// TIA Portal V19 export
FUNCTION_BLOCK "A0301_Trasporto_FB"   // FB61, LAD
TITLE = == GESTIONE NASTRI TRASPORTO ==
// stored: MemoryReserve 100, SetENOAutomatically false
   VAR_INPUT
      AreaInterface : "AreaInterface";
      ZSI : "udt_ZoneSafetyInterface";
      DSI : "udt_DeviceSafetyInterface";
      Drive : "TAx_DriveInterface";
      DataIn : "SpeedMachine_DataIn";
      CIn : Struct
         Drive : "SpeedMachine_CIn";
         OP_SemiAut_PB : Bool;
      END_STRUCT;
      Config : "SpeedMachine_Config";
      HWID_Ax_TEL1 : HW_SUBMODULE;
   END_VAR
   VAR_OUTPUT
      MachineInterface { ExternalAccessible := 'False'; ExternalVisible := 'False'; ExternalWritable := 'False'} : "MachineInterface";
      COut : Struct
         Ax : "SpeedMachine_COut";
         Ax_VelOveride : Struct
            Enable : Bool;
            Value : Real;
         END_STRUCT;
      END_STRUCT;
   END_VAR
   VAR_IN_OUT
      Par : Struct
         Ax : "SpeedMachine_Par";
         Ax_Aut : "A0301_Mach_Speed_Par";
      END_STRUCT;
   END_VAR
   VAR
      Alarm : Struct
         Ax { ExternalVisible := 'False'} : "SpeedMachine_Alr";
      END_STRUCT;
      Warning : Struct
         Ax { S7_SetPoint := 'True'} : "SpeedMachine_Wng";
         OP_REST_MissingCnd : Bool;   // Mancanza comando arresto
         OP_WORK_MissingCnd : Bool;   // Mancanza consenso lavoro
      END_STRUCT;
      Ax : "SpeedMachine_FB";
      ValueVelOvr { ExternalAccessible := 'False'; ExternalVisible := 'False'; ExternalWritable := 'False'} : Array[1..10] of Real;
      Sts : Struct
         OP_CanMoveFreely : Bool;
         OP_Bwd_Cnd : Bool;
         OP_Fwd_Cnd : Bool;
      END_STRUCT;
      Ctrl : Struct
         OP_Bwd_Man : Bool;
         OP_Fwd_Man : Bool;
         OP_Bwd_Aut : Bool;
         OP_Fwd_Aut : Bool;
         OP_Bwd_Run : Bool;
         OP_Fwd_Run : Bool;
      END_STRUCT;
      AUX : Struct
         OP_Bwd_PB : Bool;
         OP_Fwd_PB : Bool;
      END_STRUCT;
      TON_OP_REST_MissingCnd { S7_SetPoint := 'True'} : TON_TIME;
      TON_OP_WORK_MissingCnd { S7_SetPoint := 'True'} : TON_TIME;
   END_VAR
   VAR_TEMP
      PE : Struct
         OP_Bwd_PB : Bool;
         OP_Fwd_PB : Bool;
      END_STRUCT;
      VelOvr_Max : Real;   // Velocità max trovata
      i : Int;
      Check : Struct
         Cndz1_StartFwd : Bool;   // Check conditions to P4
         Cndz2_StartFwd : Bool;   // Check conditions to Allineatore laterale
      END_STRUCT;
   END_VAR
   VAR_TEMP   // added for the SCL form of the ladder/FBD networks
      _w1 : Bool;
      _w2 : Bool;
      _w3 : Bool;
   END_VAR
BEGIN

REGION Network 1 (SCL): == Riferimenti [Ax] - Speed Machine ==
   // ******************************************************************************************
   REGION // TRASFERIMENTO DELLE RAMPE

       // Rampe in Manuale
       IF #AreaInterface.Man AND NOT #CIn.OP_SemiAut_PB THEN
           #Ax.CIn.Manager.Vel := #Par.Ax.Man.VelFwdHigh;
           #Ax.CIn.Manager.Acc := #Par.Ax.Man.Acc;
           #Ax.CIn.Manager.Dec := #Par.Ax.Man.Dec;
       END_IF;
   END_REGION


   // ******************************************************************************************
   REGION // CALCOLO DELLA VELOCITA' TRASFERITA DALL'IMPIANTO IN BASE ALLA LUNGHEZZA DEL PEZZO 

       // Inizializzo variabile di appoggio controllo overide massimo a un valore basso rispetto setpoint
       IF "Sys".AuxFirstPLCCycle THEN
           #VelOvr_Max := 100.0;
       END_IF;

       // Trasferisco le varibili su un array
       #ValueVelOvr[1] := "PPrf_MAIN".ON_WORK.A0301_A0302.Trasporto.VelOvr_PLen_UpTo_1000;
       #ValueVelOvr[2] := "PPrf_MAIN".ON_WORK.A0301_A0302.Trasporto.VelOvr_PLen_UpTo_1500;
       #ValueVelOvr[3] := "PPrf_MAIN".ON_WORK.A0301_A0302.Trasporto.VelOvr_PLen_UpTo_2000;
       #ValueVelOvr[4] := "PPrf_MAIN".ON_WORK.A0301_A0302.Trasporto.VelOvr_PLen_UpTo_2500;
       #ValueVelOvr[5] := "PPrf_MAIN".ON_WORK.A0301_A0302.Trasporto.VelOvr_PLen_UpTo_3000;
       #ValueVelOvr[6] := "PPrf_MAIN".ON_WORK.A0301_A0302.Trasporto.VelOvr_PLen_UpTo_3500;
       #ValueVelOvr[7] := "PPrf_MAIN".ON_WORK.A0301_A0302.Trasporto.VelOvr_PLen_UpTo_4000;
       #ValueVelOvr[8] := "PPrf_MAIN".ON_WORK.A0301_A0302.Trasporto.VelOvr_PLen_UpTo_4500;
       #ValueVelOvr[9] := "PPrf_MAIN".ON_WORK.A0301_A0302.Trasporto.VelOvr_PLen_UpTo_5000;
       #ValueVelOvr[10] := "PPrf_MAIN".ON_WORK.A0301_A0302.Trasporto.VelOvr_PLen_UpTo_5500;


       // Ciclo per verificare la variabile maggiore per prenderla in lavoro
       FOR #i := 1 TO 10 DO
           IF #ValueVelOvr[#i] >= #VelOvr_Max THEN
               #VelOvr_Max := #ValueVelOvr[#i];
           END_IF;
       END_FOR;
   END_REGION ;

   IF #VelOvr_Max = 0.0 THEN
       #VelOvr_Max := 100.0;
   END_IF;

   // ******************************************************************************************
   REGION // CALCOLO DELLA VELOCITA' E TRASFERIMENTO IN BASE ALLO STATO IMPIANTO
       #Ax.CIn.Manager := #CIn.Drive.Manager;

       IF #Ax.CIn.Manager.Control_ON THEN
           // CALCOLO VELOCITA' IN BASE ALL'OVERIDE
           IF #Ax.AreaInterface.Aut THEN
               #Ax.CIn.Manager.Vel := (#Par.Ax_Aut.Aut_Vel * #VelOvr_Max);
           END_IF;

           IF #CIn.OP_SemiAut_PB AND NOT #Ax.AreaInterface.Aut THEN
               #Ax.CIn.Manager.Vel := (#Par.Ax_Aut.SemiAut_Vel* #VelOvr_Max);
               #Ax.CIn.Manager.Acc := #Par.Ax_Aut.Aut_Acc;
               #Ax.CIn.Manager.Dec := #Par.Ax_Aut.Aut_Dec;
           END_IF;
       END_IF;
   END_REGION ;
   //


       #COut.Ax_VelOveride.Enable := TRUE;
       #COut.Ax_VelOveride.Value := #VelOvr_Max;
END_REGION

REGION Network 3: Operazione può muoversi liberamente perchè non sposta nessun BEAM
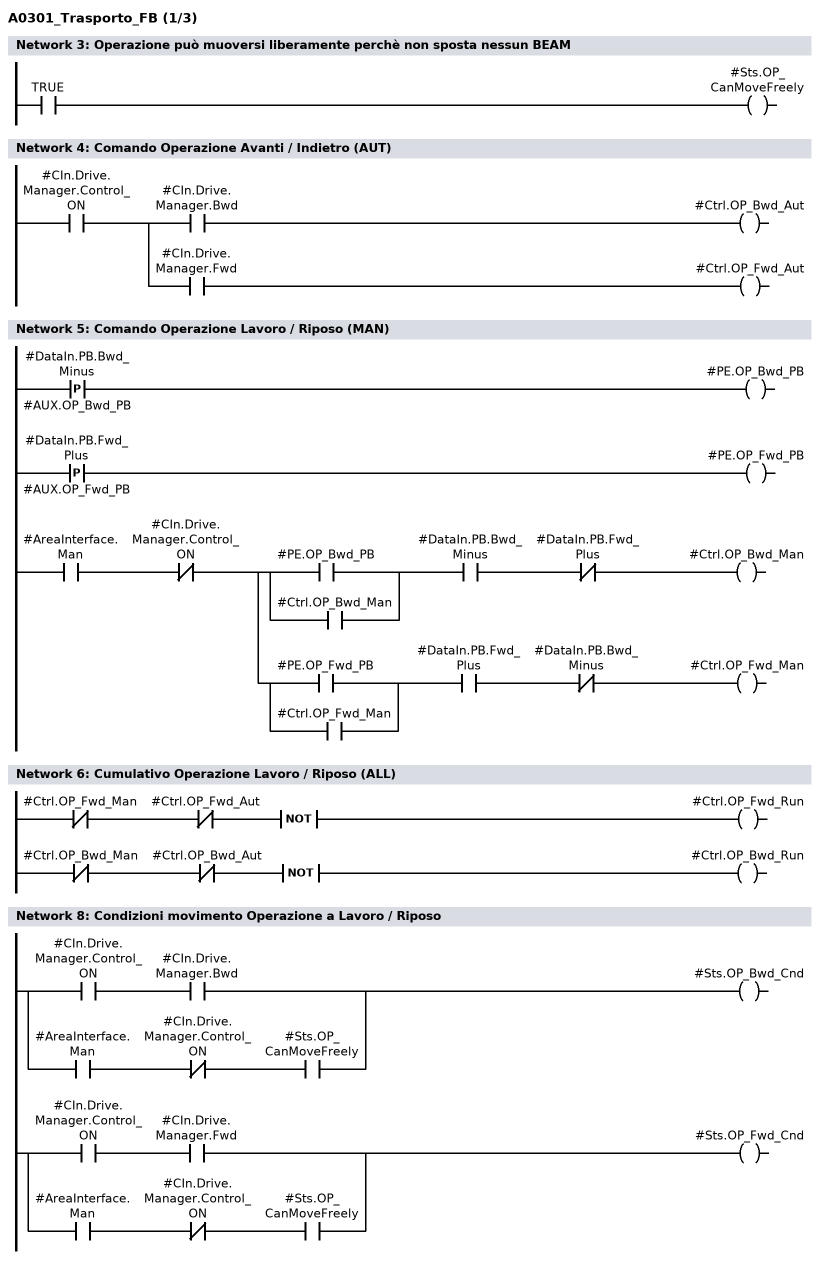
   RUNG wire#powerrail
      Contact( TRUE )
      Coil( #Sts.OP_CanMoveFreely )
   END_RUNG
   // the same network as SCL:
   #Sts.OP_CanMoveFreely := TRUE;
END_REGION

REGION Network 4: Comando Operazione Avanti / Indietro (AUT)
   RUNG wire#powerrail
      Contact( #CIn.Drive.Manager.Control_ON )
      wire#w1
      Contact( #CIn.Drive.Manager.Bwd )
      Coil( #Ctrl.OP_Bwd_Aut )
   END_RUNG
   RUNG wire#w1
      Contact( #CIn.Drive.Manager.Fwd )
      Coil( #Ctrl.OP_Fwd_Aut )
   END_RUNG
   // the same network as SCL:
   #Ctrl.OP_Bwd_Aut := #CIn.Drive.Manager.Control_ON AND #CIn.Drive.Manager.Bwd;
   #Ctrl.OP_Fwd_Aut := #CIn.Drive.Manager.Control_ON AND #CIn.Drive.Manager.Fwd;
END_REGION

REGION Network 5: Comando Operazione Lavoro / Riposo (MAN)
   RUNG wire#powerrail
      P_Contact(operand := #DataIn.PB.Bwd_Minus, bit := #AUX.OP_Bwd_PB)
      Coil( #PE.OP_Bwd_PB )
   END_RUNG
   RUNG wire#powerrail
      P_Contact(operand := #DataIn.PB.Fwd_Plus, bit := #AUX.OP_Fwd_PB)
      Coil( #PE.OP_Fwd_PB )
   END_RUNG
   RUNG wire#powerrail
      Contact( #AreaInterface.Man )
      I_Contact( #CIn.Drive.Manager.Control_ON )
      wire#w1
      Contact( #PE.OP_Bwd_PB )
      wire#w2
      Contact( #DataIn.PB.Bwd_Minus )
      I_Contact( #DataIn.PB.Fwd_Plus )
      Coil( #Ctrl.OP_Bwd_Man )
   END_RUNG
   RUNG wire#w1
      Contact( #Ctrl.OP_Bwd_Man )
   END_RUNG wire#w2
   RUNG wire#w1
      Contact( #PE.OP_Fwd_PB )
      wire#w3
      Contact( #DataIn.PB.Fwd_Plus )
      I_Contact( #DataIn.PB.Bwd_Minus )
      Coil( #Ctrl.OP_Fwd_Man )
   END_RUNG
   RUNG wire#w1
      Contact( #Ctrl.OP_Fwd_Man )
   END_RUNG wire#w3
   // the same network as SCL:
   #_w1 := #DataIn.PB.Bwd_Minus AND NOT #AUX.OP_Bwd_PB;   // rising edge of #DataIn.PB.Bwd_Minus
   #AUX.OP_Bwd_PB := #DataIn.PB.Bwd_Minus;
   #PE.OP_Bwd_PB := #_w1;
   #_w2 := #DataIn.PB.Fwd_Plus AND NOT #AUX.OP_Fwd_PB;   // rising edge of #DataIn.PB.Fwd_Plus
   #AUX.OP_Fwd_PB := #DataIn.PB.Fwd_Plus;
   #PE.OP_Fwd_PB := #_w2;
   #_w3 := #AreaInterface.Man AND NOT #CIn.Drive.Manager.Control_ON;
   #Ctrl.OP_Bwd_Man := #_w3 AND (#PE.OP_Bwd_PB OR #Ctrl.OP_Bwd_Man) AND #DataIn.PB.Bwd_Minus AND NOT #DataIn.PB.Fwd_Plus;
   #Ctrl.OP_Fwd_Man := #_w3 AND (#PE.OP_Fwd_PB OR #Ctrl.OP_Fwd_Man) AND #DataIn.PB.Fwd_Plus AND NOT #DataIn.PB.Bwd_Minus;
END_REGION

REGION Network 6: Cumulativo Operazione Lavoro / Riposo (ALL)
   RUNG wire#powerrail
      I_Contact( #Ctrl.OP_Fwd_Man )
      I_Contact( #Ctrl.OP_Fwd_Aut )
      Not()
      Coil( #Ctrl.OP_Fwd_Run )
   END_RUNG
   RUNG wire#powerrail
      I_Contact( #Ctrl.OP_Bwd_Man )
      I_Contact( #Ctrl.OP_Bwd_Aut )
      Not()
      Coil( #Ctrl.OP_Bwd_Run )
   END_RUNG
   // the same network as SCL:
   #Ctrl.OP_Fwd_Run := NOT (NOT #Ctrl.OP_Fwd_Man AND NOT #Ctrl.OP_Fwd_Aut);
   #Ctrl.OP_Bwd_Run := NOT (NOT #Ctrl.OP_Bwd_Man AND NOT #Ctrl.OP_Bwd_Aut);
END_REGION

REGION Network 7: <+>
END_REGION

REGION Network 8: Condizioni movimento Operazione a Lavoro / Riposo
   RUNG wire#powerrail
      Contact( #CIn.Drive.Manager.Control_ON )
      Contact( #CIn.Drive.Manager.Bwd )
      wire#w1
      Coil( #Sts.OP_Bwd_Cnd )
   END_RUNG
   RUNG wire#powerrail
      Contact( #AreaInterface.Man )
      I_Contact( #CIn.Drive.Manager.Control_ON )
      Contact( #Sts.OP_CanMoveFreely )
   END_RUNG wire#w1
   RUNG wire#powerrail
      Contact( #CIn.Drive.Manager.Control_ON )
      Contact( #CIn.Drive.Manager.Fwd )
      wire#w2
      Coil( #Sts.OP_Fwd_Cnd )
   END_RUNG
   RUNG wire#powerrail
      Contact( #AreaInterface.Man )
      I_Contact( #CIn.Drive.Manager.Control_ON )
      Contact( #Sts.OP_CanMoveFreely )
   END_RUNG wire#w2
   // the same network as SCL:
   #Sts.OP_Bwd_Cnd := (#CIn.Drive.Manager.Control_ON AND #CIn.Drive.Manager.Bwd) OR (#AreaInterface.Man AND NOT #CIn.Drive.Manager.Control_ON AND #Sts.OP_CanMoveFreely);
   #Sts.OP_Fwd_Cnd := (#CIn.Drive.Manager.Control_ON AND #CIn.Drive.Manager.Fwd) OR (#AreaInterface.Man AND NOT #CIn.Drive.Manager.Control_ON AND #Sts.OP_CanMoveFreely);
END_REGION

REGION Network 9 (SCL): [Ax] Cin Manager Comando arresto / lavoro
   //
   #Ax.CIn.Manager.Bwd := FALSE;
   //************************************
   #Ax.CIn.Manager.Fwd := FALSE;
   //
   // CIn Manager  Control ON se ho un richiesta di comando attiva
   #Ax.CIn.Manager.Control_ON := #Ctrl.OP_Fwd_Run OR #Ctrl.OP_Bwd_Run;

   // CIn Manager Frw se ho un richiesta di comando arresto attiva
   #Ax.CIn.Manager.Fwd := #Ctrl.OP_Fwd_Run AND #Sts.OP_Fwd_Cnd ;

   // CIn Manager Brw se ho un richiesta di comando arresto attiva
   #Ax.CIn.Manager.Bwd := #Ctrl.OP_Bwd_Run AND #Sts.OP_Bwd_Cnd;
END_REGION

REGION Network 10 (SCL): [Ax] CIn Abilitazioni Stop Manager
   // CIn Manager Stop per richiesta apertura safety
   // 
   #Ax.CIn.Manager.EnableStopDoorOpeningReq := #CIn.Drive.Manager.EnableStopDoorOpeningReq;

   // CIn Manager Stop in fase delle macchine precedenti
   // 
   #Ax.CIn.Manager.EnableStopInPhase := #CIn.Drive.Manager.EnableStopInPhase;

   // CIn Manager Stop programmato configurabile a piacere
   // 
   #Ax.CIn.Manager.EnableStopProgrammed := #CIn.Drive.Manager.EnableStopProgrammed;
END_REGION

REGION Network 11: <+>
END_REGION

REGION Network 12: Warning manacanza condizioni esecuzione Operazione RIPOSO / LAVORO
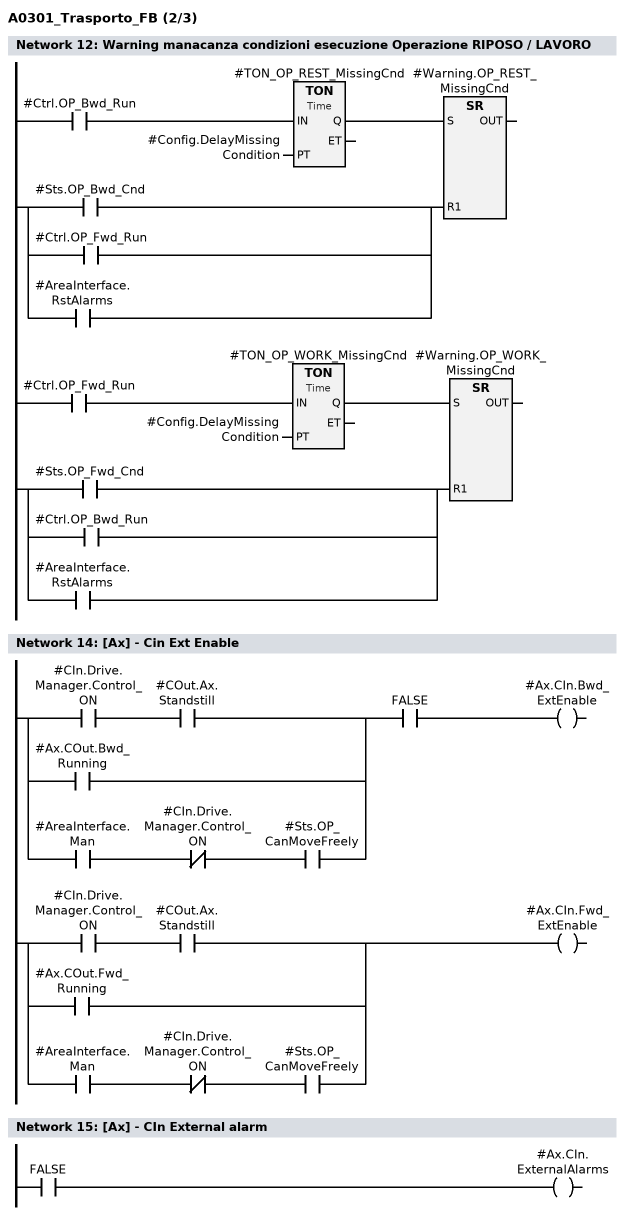
   RUNG wire#powerrail
      Contact( #Ctrl.OP_Bwd_Run )
      { S7_Templates := "time_type := Time" } #TON_OP_REST_MissingCnd.TON(pt := #Config.DelayMissingCondition, et =>)
      S_SR(operand := #Warning.OP_REST_MissingCnd, r1 := wire#w1)
   END_RUNG
   RUNG wire#powerrail
      Contact( #Sts.OP_Bwd_Cnd )
   END_RUNG wire#w1
   RUNG wire#powerrail
      Contact( #Ctrl.OP_Fwd_Run )
   END_RUNG wire#w1
   RUNG wire#powerrail
      Contact( #AreaInterface.RstAlarms )
   END_RUNG wire#w1
   RUNG wire#powerrail
      Contact( #Ctrl.OP_Fwd_Run )
      { S7_Templates := "time_type := Time" } #TON_OP_WORK_MissingCnd.TON(pt := #Config.DelayMissingCondition, et =>)
      S_SR(operand := #Warning.OP_WORK_MissingCnd, r1 := wire#w2)
   END_RUNG
   RUNG wire#powerrail
      Contact( #Sts.OP_Fwd_Cnd )
   END_RUNG wire#w2
   RUNG wire#powerrail
      Contact( #Ctrl.OP_Bwd_Run )
   END_RUNG wire#w2
   RUNG wire#powerrail
      Contact( #AreaInterface.RstAlarms )
   END_RUNG wire#w2
   // the same network as SCL:
   #TON_OP_REST_MissingCnd(IN := #Ctrl.OP_Bwd_Run, PT := #Config.DelayMissingCondition);   // TON
   IF #TON_OP_REST_MissingCnd.Q THEN
       #Warning.OP_REST_MissingCnd := TRUE;   // SR flip-flop
   END_IF;
   IF #Sts.OP_Bwd_Cnd OR #Ctrl.OP_Fwd_Run OR #AreaInterface.RstAlarms THEN
       #Warning.OP_REST_MissingCnd := FALSE;
   END_IF;
   #TON_OP_WORK_MissingCnd(IN := #Ctrl.OP_Fwd_Run, PT := #Config.DelayMissingCondition);   // TON
   IF #TON_OP_WORK_MissingCnd.Q THEN
       #Warning.OP_WORK_MissingCnd := TRUE;   // SR flip-flop
   END_IF;
   IF #Sts.OP_Fwd_Cnd OR #Ctrl.OP_Bwd_Run OR #AreaInterface.RstAlarms THEN
       #Warning.OP_WORK_MissingCnd := FALSE;
   END_IF;
END_REGION

REGION Network 13: <+>
END_REGION

REGION Network 14: [Ax] - Cin Ext Enable
   RUNG wire#powerrail
      Contact( #CIn.Drive.Manager.Control_ON )
      Contact( #COut.Ax.Standstill )
      wire#w1
      Contact( FALSE )
      Coil( #Ax.CIn.Bwd_ExtEnable )
   END_RUNG
   RUNG wire#powerrail
      Contact( #Ax.COut.Bwd_Running )
   END_RUNG wire#w1
   RUNG wire#powerrail
      Contact( #AreaInterface.Man )
      I_Contact( #CIn.Drive.Manager.Control_ON )
      Contact( #Sts.OP_CanMoveFreely )
   END_RUNG wire#w1
   RUNG wire#powerrail
      Contact( #CIn.Drive.Manager.Control_ON )
      Contact( #COut.Ax.Standstill )
      wire#w2
      Coil( #Ax.CIn.Fwd_ExtEnable )
   END_RUNG
   RUNG wire#powerrail
      Contact( #Ax.COut.Fwd_Running )
   END_RUNG wire#w2
   RUNG wire#powerrail
      Contact( #AreaInterface.Man )
      I_Contact( #CIn.Drive.Manager.Control_ON )
      Contact( #Sts.OP_CanMoveFreely )
   END_RUNG wire#w2
   // the same network as SCL:
   #Ax.CIn.Bwd_ExtEnable := ((#CIn.Drive.Manager.Control_ON AND #COut.Ax.Standstill) OR #Ax.COut.Bwd_Running OR (#AreaInterface.Man AND NOT #CIn.Drive.Manager.Control_ON AND #Sts.OP_CanMoveFreely)) AND FALSE;
   #Ax.CIn.Fwd_ExtEnable := (#CIn.Drive.Manager.Control_ON AND #COut.Ax.Standstill) OR #Ax.COut.Fwd_Running OR (#AreaInterface.Man AND NOT #CIn.Drive.Manager.Control_ON AND #Sts.OP_CanMoveFreely);
END_REGION

REGION Network 15: [Ax] - CIn External alarm
   RUNG wire#powerrail
      Contact( FALSE )
      Coil( #Ax.CIn.ExternalAlarms )
   END_RUNG
   // the same network as SCL:
   #Ax.CIn.ExternalAlarms := FALSE;
END_REGION

REGION Network 16: <+>
END_REGION

REGION Network 17: [Ax] - SpeedMachine
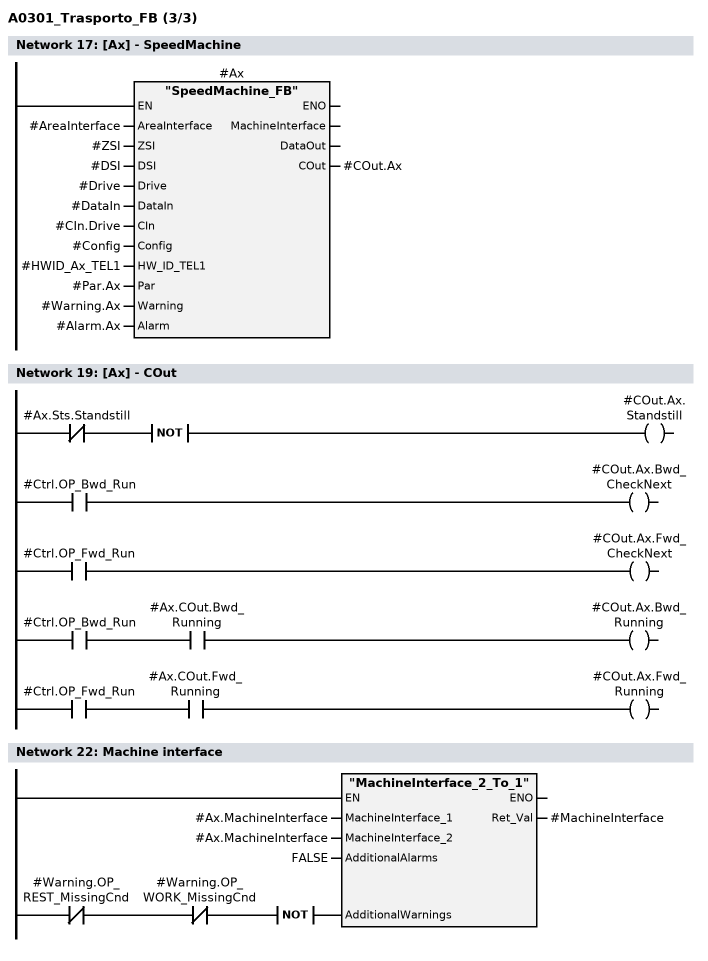
   RUNG wire#powerrail
      #Ax(AreaInterface := #AreaInterface, ZSI := #ZSI, DSI := #DSI, Drive := #Drive, DataIn := #DataIn, CIn := #CIn.Drive, Config := #Config, HW_ID_TEL1 := #HWID_Ax_TEL1, Par := #Par.Ax, Warning := #Warning.Ax, Alarm := #Alarm.Ax, MachineInterface =>, DataOut =>, COut => #COut.Ax)
   END_RUNG
   // the same network as SCL:
   #Ax(AreaInterface := #AreaInterface,   // "SpeedMachine_FB"
       ZSI := #ZSI,
       DSI := #DSI,
       Drive := #Drive,
       DataIn := #DataIn,
       CIn := #CIn.Drive,
       Config := #Config,
       HW_ID_TEL1 := #HWID_Ax_TEL1,
       Par := #Par.Ax,
       Warning := #Warning.Ax,
       Alarm := #Alarm.Ax,
       COut => #COut.Ax);
END_REGION

REGION Network 18: <+>
END_REGION

REGION Network 19: [Ax] - COut
   RUNG wire#powerrail
      I_Contact( #Ax.Sts.Standstill )
      Not()
      Coil( #COut.Ax.Standstill )
   END_RUNG
   RUNG wire#powerrail
      Contact( #Ctrl.OP_Bwd_Run )
      Coil( #COut.Ax.Bwd_CheckNext )
   END_RUNG
   RUNG wire#powerrail
      Contact( #Ctrl.OP_Fwd_Run )
      Coil( #COut.Ax.Fwd_CheckNext )
   END_RUNG
   RUNG wire#powerrail
      Contact( #Ctrl.OP_Bwd_Run )
      Contact( #Ax.COut.Bwd_Running )
      Coil( #COut.Ax.Bwd_Running )
   END_RUNG
   RUNG wire#powerrail
      Contact( #Ctrl.OP_Fwd_Run )
      Contact( #Ax.COut.Fwd_Running )
      Coil( #COut.Ax.Fwd_Running )
   END_RUNG
   // the same network as SCL:
   #COut.Ax.Standstill := NOT (NOT #Ax.Sts.Standstill);
   #COut.Ax.Bwd_CheckNext := #Ctrl.OP_Bwd_Run;
   #COut.Ax.Fwd_CheckNext := #Ctrl.OP_Fwd_Run;
   #COut.Ax.Bwd_Running := #Ctrl.OP_Bwd_Run AND #Ax.COut.Bwd_Running;
   #COut.Ax.Fwd_Running := #Ctrl.OP_Fwd_Run AND #Ax.COut.Fwd_Running;
END_REGION

REGION Network 21: << MAIN MACHINE STATUS >>
END_REGION

REGION Network 22: Machine interface
   RUNG wire#powerrail
      "MachineInterface_2_To_1"(AdditionalWarnings := wire#w1, MachineInterface_1 := #Ax.MachineInterface, MachineInterface_2 := #Ax.MachineInterface, AdditionalAlarms := FALSE, Ret_Val => #MachineInterface)
   END_RUNG
   RUNG wire#powerrail
      I_Contact( #Warning.OP_REST_MissingCnd )
      I_Contact( #Warning.OP_WORK_MissingCnd )
      Not()
   END_RUNG wire#w1
   // the same network as SCL:
   #MachineInterface := "MachineInterface_2_To_1"(MachineInterface_1 := #Ax.MachineInterface,
                           MachineInterface_2 := #Ax.MachineInterface,
                           AdditionalAlarms := FALSE,
                           AdditionalWarnings := NOT (NOT #Warning.OP_REST_MissingCnd AND NOT #Warning.OP_WORK_MissingCnd));
END_REGION
END_FUNCTION_BLOCK
